FUNCTION_BLOCK motor
VAR_INPUT
	rotateForward: BOOL;
	rotateBackward: BOOL;
END_VAR
VAR_OUTPUT
	direction: BOOL;
	movement: BOOL;
END_VAR

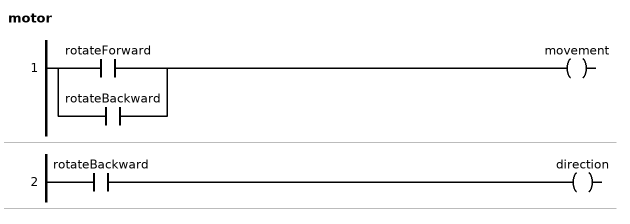
// NETWORK 1
movement := rotateForward OR rotateBackward;

// NETWORK 2
direction := rotateBackward;

END_FUNCTION_BLOCK

(* stored: Version 1.1.0.1, ProductVersion 3.1.4024.13
   POU motor: Id {480415d5-26d5-41ab-a4b3-a97377ecb90d}, SpecialFunc None *)
